ABB RAPID module: 000BBA84

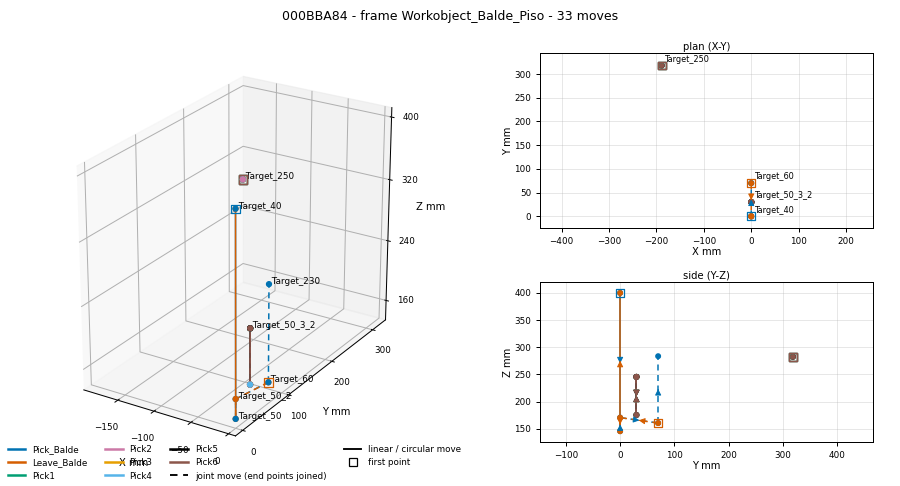
[picture p0: tool path of 000BBA84 in frame Workobject_Balde_Piso, 33 of 59 moves have a stored position in this frame; points joined in program order, loops and branches not executed]
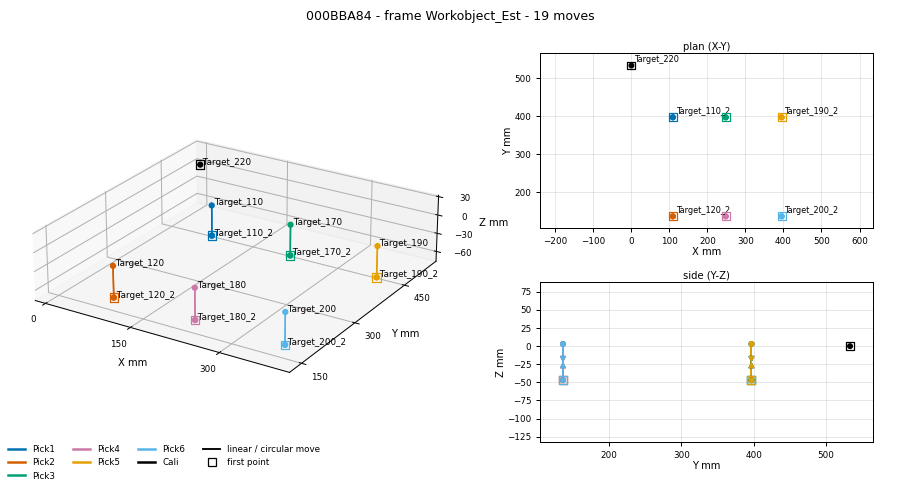
[picture p1: tool path of 000BBA84 in frame Workobject_Est, 19 of 59 moves have a stored position in this frame; points joined in program order, loops and branches not executed]
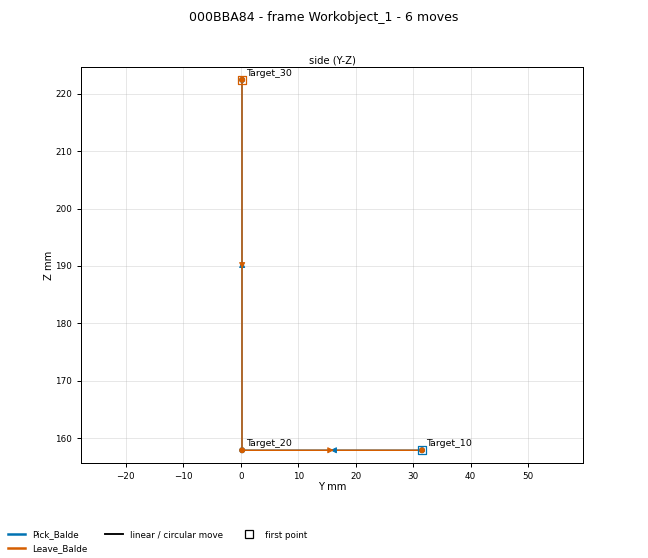
[picture p2: tool path of 000BBA84 in frame Workobject_1, 6 of 59 moves have a stored position in this frame; points joined in program order, loops and branches not executed]
MODULE Module1
	CONST robtarget Target_10:=[[-0.541791285,31.542690631,157.927772118],[0.338220375,0.61994805,0.62152642,-0.339081557],[-1,1,-1,0],[9E+09,9E+09,9E+09,9E+09,9E+09,9E+09]];
	CONST robtarget Target_20:=[[-0.54180672,0.235098408,157.927793799],[0.499363871,0.499363893,0.500635292,-0.500635328],[-1,1,-2,0],[9E+09,9E+09,9E+09,9E+09,9E+09,9E+09]];
	CONST robtarget Target_30:=[[-0.541814528,0.23509908,222.389598203],[0.499363884,0.49936382,0.500635317,-0.500635363],[-1,1,-2,0],[9E+09,9E+09,9E+09,9E+09,9E+09,9E+09]];
	CONST robtarget Target_40:=[[0,0,400],[0.499363884,0.49936382,0.500635317,-0.500635363],[0,1,-3,0],[9E+09,9E+09,9E+09,9E+09,9E+09,9E+09]];
	CONST robtarget Target_50:=[[-0.038127492,-0.000030739,145.519742619],[0.499363836,0.499363825,0.500635306,-0.500635416],[-1,2,-3,0],[9E+09,9E+09,9E+09,9E+09,9E+09,9E+09]];
	CONST robtarget Target_60:=[[0,70,160.52],[0.182019153,0.682470244,0.683552682,-0.184008491],[0,2,-2,0],[9E+09,9E+09,9E+09,9E+09,9E+09,9E+09]];
    CONST robtarget Target_70:=[[605.229348481,0,514.125118395],[0.275637355,0,0.961261696,0],[0,0,0,0],[9E+09,9E+09,9E+09,9E+09,9E+09,9E+09]];
    CONST robtarget Target_90:=[[204.199229947,-72.229383295,-619.023797732],[0.618449546,0.618449531,0.34281213,0.342812167],[0,-2,1,0],[9E+09,9E+09,9E+09,9E+09,9E+09,9E+09]];
    CONST robtarget Target_80:=[[-77.125218661,-72.22939491,-596.502903487],[0.618449548,0.618449544,0.342812142,0.342812128],[0,-1,0,0],[9E+09,9E+09,9E+09,9E+09,9E+09,9E+09]];
    CONST robtarget Target_50_2:=[[-0.038127492,-0.000030739,170.519742619],[0.182018295,0.682471059,0.683552878,-0.184005593],[-1,1,-2,0],[9E+09,9E+09,9E+09,9E+09,9E+09,9E+09]];
	CONST robtarget Target_160:=[[605.229348481,0,514.125118395],[0.275637355,0,0.961261696,0],[0,0,0,0],[9E+09,9E+09,9E+09,9E+09,9E+09,9E+09]];
	CONST robtarget Target_130:=[[108.313469676,92.052338402,147.49758099],[0.444719526,0.257906476,0.743119571,0.428348101],[0,-2,-2,0],[9E+09,9E+09,9E+09,9E+09,9E+09,9E+09]];
	CONST robtarget Target_110_2:=[[109,396.75,-47],[1,0,0,0],[0,2,-2,0],[9E+09,9E+09,9E+09,9E+09,9E+09,9E+09]];
	CONST robtarget Target_110:=[[109,396.75,3],[1,0,0,0],[0,2,-2,0],[9E+09,9E+09,9E+09,9E+09,9E+09,9E+09]];
	CONST robtarget Target_50_3_2:=[[0.216181367,29.999981348,245.519415627],[0.611593294,0.353103544,0.613150552,-0.354002726],[0,-3,2,0],[9E+09,9E+09,9E+09,9E+09,9E+09,9E+09]];
	CONST robtarget Target_150:=[[0.216193734,29.999948387,175.359992959],[0.611593362,0.353103485,0.613150461,-0.354002825],[0,-2,1,0],[9E+09,9E+09,9E+09,9E+09,9E+09,9E+09]];
	CONST robtarget Target_120_2:=[[109,136.25,-47],[1,0,0,0],[0,1,-2,0],[9E+09,9E+09,9E+09,9E+09,9E+09,9E+09]];
	CONST robtarget Target_120:=[[109,136.25,3],[1,0,0,0],[0,1,-2,0],[9E+09,9E+09,9E+09,9E+09,9E+09,9E+09]];
	CONST robtarget Target_170_2:=[[248,396.75,-47],[0.216439613,0,0,0.976296007],[0,2,-2,0],[9E+09,9E+09,9E+09,9E+09,9E+09,9E+09]];
	CONST robtarget Target_170:=[[248,396.75,3],[0.216439613,0,0,0.976296007],[0,2,-2,0],[9E+09,9E+09,9E+09,9E+09,9E+09,9E+09]];
	CONST robtarget Target_180_2:=[[248,136.25,-47],[0.707106781,0,0,0.707106781],[0,1,-2,0],[9E+09,9E+09,9E+09,9E+09,9E+09,9E+09]];
	CONST robtarget Target_180:=[[248,136.25,3],[0.707106781,0,0,0.707106781],[0,1,-2,0],[9E+09,9E+09,9E+09,9E+09,9E+09,9E+09]];
	CONST robtarget Target_190_2:=[[395,396.75,-47],[0.382683432,0,0,0.923879533],[0,2,-2,0],[9E+09,9E+09,9E+09,9E+09,9E+09,9E+09]];
	CONST robtarget Target_190:=[[395,396.75,3],[0.382683432,0,0,0.923879533],[0,2,-2,0],[9E+09,9E+09,9E+09,9E+09,9E+09,9E+09]];
	CONST robtarget Target_200_2:=[[395,136.25,-47],[0.707106781,0,0,0.707106781],[0,1,-2,0],[9E+09,9E+09,9E+09,9E+09,9E+09,9E+09]];
	CONST robtarget Target_200:=[[395,136.25,3],[0.707106781,0,0,0.707106781],[0,1,-2,0],[9E+09,9E+09,9E+09,9E+09,9E+09,9E+09]];
	CONST robtarget Target_60_2:=[[0,70,280.52],[0.182019153,0.682470244,0.683552682,-0.184008491],[0,-2,-2,0],[9E+09,9E+09,9E+09,9E+09,9E+09,9E+09]];
	CONST robtarget Target_210:=[[108.31348361,92.052306653,267.497558788],[0.444719566,0.257906454,0.743119625,0.428347979],[0,-2,-2,0],[9E+09,9E+09,9E+09,9E+09,9E+09,9E+09]];
	CONST robtarget Target_220:=[[0,533,0],[1,0,0,0],[1,2,2,0],[9E+09,9E+09,9E+09,9E+09,9E+09,9E+09]];
    CONST robtarget Target_250:=[[-188.843410439,317.985657737,282.635376599],[0.28601825,0.002111346,-0.703849705,-0.650218959],[0,1,-1,0],[9E+09,9E+09,9E+09,9E+09,9E+09,9E+09]];
    CONST robtarget Target_230:=[[0.000068646,70.00001103,283.574285968],[0.182019117,0.682470266,0.683552671,-0.184008489],[0,2,-2,0],[9E+09,9E+09,9E+09,9E+09,9E+09,9E+09]];
    CONST  speeddata vel := v500;
    !***********************************************************
    !
    ! Module:  Module1
    !
    ! Description:
    !   <Insert description here>
    !
    ! Author: maaro
    !
    ! Version: 1.0
    !
    !***********************************************************


    !***********************************************************
    !
    ! Procedure main
    !
    !   This is the entry point of your program
    !
    !***********************************************************
    PROC main()
        Go_Home;
        Pick_Balde;
        Pick1;
        Pick2;
        Pick3;
        Leave_Balde;
        Go_Home;
    ENDPROC
    PROC Pick_Balde()
        MoveJ Target_10,vel,z100,TD_Hook\WObj:=Workobject_1;
        MoveL Target_20,vel,fine,TD_Hook\WObj:=Workobject_1;
        !PulseDO att_Balde;
        WaitTime 0.5;
        MoveL Target_30,v200,z100,TD_Hook\WObj:=Workobject_1;
        MoveL Target_40,v200,fine,TD_Hook\WObj:=Workobject_Balde_Piso;
        WaitTime 1;
        MoveL Target_50,v200,fine,TD_Hook\WObj:=Workobject_Balde_Piso;
        !PulseDO det_Balde;
        WaitTime 0.5;
        MoveJ Target_50_2,v50,fine,TD_Hook\WObj:=Workobject_Balde_Piso;
        MoveJ Target_60,vel,z10,TD_Hook\WObj:=Workobject_Balde_Piso;
		MoveJ Target_230,vel,z5,TD_Hook\WObj:=Workobject_Balde_Piso;
    ENDPROC
    PROC Leave_Balde()
        MoveJ Target_60,vel,fine,TD_Hook\WObj:=Workobject_Balde_Piso;
        MoveJ Target_50_2,v50,z10,TD_Hook\WObj:=Workobject_Balde_Piso;
        MoveJ Target_50,v50,fine,TD_Hook\WObj:=Workobject_Balde_Piso;
        !PulseDO att_Balde;
        WaitTime 0.5;
        MoveL Target_40,vel,z150,TD_Hook\WObj:=Workobject_Balde_Piso;
        MoveL Target_30,vel,z100,TD_Hook\WObj:=Workobject_1;
        MoveL Target_20,v100,fine,TD_Hook\WObj:=Workobject_1;
        !PulseDO det_Balde;
        WaitTime 0.5;
        MoveL Target_10,vel,z100,TD_Hook\WObj:=Workobject_1;
    ENDPROC
    PROC Go_Home()
        MoveJ Target_160,vel,z0,TD_SuctionPad\WObj:=wobj0;
    ENDPROC
	PROC Pick1()
	    MoveJ Target_250,vel,z5,TD_SuctionPad\WObj:=Workobject_Balde_Piso;
	    MoveJ Target_110_2,vel,z5,TD_SuctionPad\WObj:=Workobject_Est;
        PulseDO DO_02;
	    MoveL Target_110,v50,fine,TD_SuctionPad\WObj:=Workobject_Est;
	    !PulseDO att_Pieza2;
	    WaitTime 1;
	    MoveL Target_110_2,vel,z100,TD_SuctionPad\WObj:=Workobject_Est;
	    MoveJ Target_50_3_2,vel,z5,TD_SuctionPad\WObj:=Workobject_Balde_Piso;
	    MoveL Target_150,vel,fine,TD_SuctionPad\WObj:=Workobject_Balde_Piso;
	    !PulseDO Det_Pieza2;
        PulseDO DO_01;
	    WaitTime 1;
        MoveJ Target_50_3_2,vel,z5,TD_SuctionPad\WObj:=Workobject_Balde_Piso;
	ENDPROC
	PROC Pick2()
	    MoveJ Target_250,vel,z5,TD_SuctionPad\WObj:=Workobject_Balde_Piso;
	    MoveJ Target_120_2,vel,z5,TD_SuctionPad\WObj:=Workobject_Est;
        PulseDO DO_02;
	    MoveL Target_120,v50,fine,TD_SuctionPad\WObj:=Workobject_Est;
	    !PulseDO att_Pieza1;
	    WaitTime 1;
	    MoveL Target_120_2,v50,z10,TD_SuctionPad\WObj:=Workobject_Est;
	    MoveJ Target_50_3_2,vel,z50,TD_SuctionPad\WObj:=Workobject_Balde_Piso;
	    MoveL Target_150,v50,fine,TD_SuctionPad\WObj:=Workobject_Balde_Piso;
        PulseDO DO_01;
	    !PulseDO Det_Pieza1;
	    WaitTime 1;
        MoveJ Target_50_3_2,vel,z50,TD_SuctionPad\WObj:=Workobject_Balde_Piso;
	ENDPROC
	PROC Pick3()
	    MoveJ Target_250,vel,z5,TD_SuctionPad\WObj:=Workobject_Balde_Piso;
	    MoveJ Target_170_2,vel,z5,TD_SuctionPad\WObj:=Workobject_Est;
        PulseDO DO_02;
	    MoveL Target_170,v50,fine,TD_SuctionPad\WObj:=Workobject_Est;
	    !PulseDO att_Pieza3;
	    WaitTime 1;
	    MoveL Target_170_2,v50,z10,TD_SuctionPad\WObj:=Workobject_Est;
	    MoveJ Target_50_3_2,vel,z50,TD_SuctionPad\WObj:=Workobject_Balde_Piso;
	    MoveL Target_150,v50,fine,TD_SuctionPad\WObj:=Workobject_Balde_Piso;
	    !PulseDO Det_Pieza3;
        PulseDO DO_01;
	    WaitTime 1;
        MoveJ Target_50_3_2,vel,z50,TD_SuctionPad\WObj:=Workobject_Balde_Piso;
	ENDPROC
	PROC Pick4()
	    MoveJ Target_250,vel,z5,TD_SuctionPad\WObj:=Workobject_Balde_Piso;
	    MoveJ Target_180_2,vel,z5,TD_SuctionPad\WObj:=Workobject_Est;
        PulseDO DO_02;
	    MoveL Target_180,v50,fine,TD_SuctionPad\WObj:=Workobject_Est;
	    !PulseDO att_Pieza4;
	    WaitTime 1;
	    MoveL Target_180_2,v50,z10,TD_SuctionPad\WObj:=Workobject_Est;
	    MoveJ Target_50_3_2,vel,z50,TD_SuctionPad\WObj:=Workobject_Balde_Piso;
	    MoveL Target_150,v50,fine,TD_SuctionPad\WObj:=Workobject_Balde_Piso;
        PulseDO DO_01;
	    !PulseDO Det_Pieza4;
	    WaitTime 1;
        MoveJ Target_50_3_2,vel,z50,TD_SuctionPad\WObj:=Workobject_Balde_Piso;
	ENDPROC
	PROC Pick5()
	    MoveJ Target_250,vel,z5,TD_SuctionPad\WObj:=Workobject_Balde_Piso;
	    MoveJ Target_190_2,vel,z5,TD_SuctionPad\WObj:=Workobject_Est;
        PulseDO DO_02;
	    MoveL Target_190,v50,fine,TD_SuctionPad\WObj:=Workobject_Est;
	    !PulseDO att_Pieza5;
	    WaitTime 1;
	    MoveL Target_190_2,v50,z10,TD_SuctionPad\WObj:=Workobject_Est;
	    MoveJ Target_50_3_2,vel,z50,TD_SuctionPad\WObj:=Workobject_Balde_Piso;
	    MoveL Target_150,v50,fine,TD_SuctionPad\WObj:=Workobject_Balde_Piso;
        PulseDO DO_01;
	    !PulseDO Det_Pieza5;
	    WaitTime 1;
        MoveJ Target_50_3_2,vel,z50,TD_SuctionPad\WObj:=Workobject_Balde_Piso;
	ENDPROC
	PROC Pick6()
	    MoveJ Target_250,vel,z5,TD_SuctionPad\WObj:=Workobject_Balde_Piso;
	    MoveJ Target_200_2,vel,z5,TD_SuctionPad\WObj:=Workobject_Est;
        PulseDO DO_02;
	    MoveL Target_200,v50,fine,TD_SuctionPad\WObj:=Workobject_Est;
	    !PulseDO att_Pieza6;
	    WaitTime 1;
	    MoveL Target_200_2,v50,z10,TD_SuctionPad\WObj:=Workobject_Est;
	    MoveJ Target_50_3_2,vel,z50,TD_SuctionPad\WObj:=Workobject_Balde_Piso;
	    MoveL Target_150,v50,fine,TD_SuctionPad\WObj:=Workobject_Balde_Piso;
        PulseDO DO_01;
	    !PulseDO Det_Pieza6;
	    WaitTime 1;
        MoveJ Target_50_3_2,vel,z50,TD_SuctionPad\WObj:=Workobject_Balde_Piso;
	ENDPROC
	PROC Cali()
	    MoveJ Target_220,v200,z5,TD_SuctionPad\WObj:=Workobject_Est;
	ENDPROC
ENDMODULE
